TYPE ST_Integrated2 :
STRUCT
	bBool			:BOOL;
	iData			:INT;
	rData			:REAL;
	sStr			:STRING;	
END_STRUCT
END_TYPE

(* stored: Version 1.1.0.1, ProductVersion 3.1.4024.15
   DUT ST_Integrated2: Id {6630e654-43ac-4cc7-a405-50d23e6dc710} *)
